// TwinCAT 3 PLC project Untitled1
// ProgramVersion: 3.1.4023.0
// libraries:
//   Tc2_Standard, * (Beckhoff Automation GmbH)
//   Tc2_System, * (Beckhoff Automation GmbH)
//   Tc3_Module, * (Beckhoff Automation GmbH)
// project tree:
//   / PlcTask.TcTTO
//   POUs/ MAIN.TcPOU (not stored)
//   TASK1/ G_Task1.TcGVL, P_Task1.TcPOU (not stored), SensorBrand.TcDUT (not stored)
//   TASK2/ F_DegToRad.TcPOU, F_UpdateParameter2.TcPOU, G_Task2.TcGVL, F_UpdateParameter.TcPOU, P_Task2.TcPOU, ST_MotorParameters.TcDUT, ST_Timer.TcDUT

CONFIGURATION Untitled1
    RESOURCE PLC ON TwinCAT3
        TASK PlcTask(INTERVAL := T#10ms, PRIORITY := 20);
        PROGRAM MAIN WITH PlcTask : MAIN;
    END_RESOURCE
END_CONFIGURATION

// ---- TASK2/ST_MotorParameters.TcDUT
TYPE ST_MotorParameters :
STRUCT
	fMaxMotorSpeed:REAL;
	fMinMotorSpeed:REAL;
END_STRUCT
END_TYPE

// ---- TASK2/ST_Timer.TcDUT
TYPE ST_Timer :
STRUCT
bTimerStart:BOOL;
tTimer:TIME;
bTimerOn:BOOL;
tEllapsedTime:TIME;
END_STRUCT
END_TYPE

// ---- TASK1/G_Task1.TcGVL
{attribute 'qualified_only'}
VAR_GLOBAL
dtvariable:DATE_AND_TIME:=DT#2023-02-07-14:01:20;

tTid:TIME:=T#5S;
aDatoArray:ARRAY[1..4]OF DATE:=[D#2023-02-07, D#2023-02-08,D#2023-02-09,D#2023-02-10];
eSensor1:SensorBrand;
bTimerStart:BOOL;
tTimer:TIME:=T#10S;
bTimerOn:BOOL;
tEllapsedTime:TIME;
END_VAR

// ---- TASK2/G_Task2.TcGVL
{attribute 'qualified_only'}
VAR_GLOBAL
	stTimer2 : ST_Timer:=(tTimer:=T#5S);
	fMotorPosDeg:REAL;
	fMototPosRad:REAL;
	stMotorParametrs:ST_MotorParameters;
	stMotorParameters2:ST_MotorParameters;
	
END_VAR

// ---- TASK2/F_DegToRad.TcPOU
FUNCTION F_DegToRad : REAL
VAR_INPUT
	fDegree:LREAL;
END_VAR
VAR
END_VAR

F_DegToRad:=fDegree*(3.14/180);

END_FUNCTION

// ---- TASK2/F_UpdateParameter2.TcPOU
FUNCTION F_UpdateParameter2 
VAR_INPUT
	bUpdateValue:BOOL;
	fNewValue:REAL;
	stMotorParameter:REFERENCE TO ST_MotorParameters;
END_VAR
VAR
END_VAR

IF bUpdateValue THEN
	stMotorParameter.fMaxMotorSpeed:=fNewValue;
ELSE
	stMotorParameter.fMaxMotorSpeed:=stMotorParameter.fMaxMotorSpeed;
END_IF

END_FUNCTION

// ---- TASK2/F_UpdateParameter.TcPOU
FUNCTION F_UpdateParameter 
VAR_INPUT
	bUpdateValue:BOOL;
	fNewValue:REAL;
	stMotorParameter:ST_MotorParameters;
END_VAR
VAR
END_VAR

IF bUpdateValue THEN
	stMotorParameter.fMaxMotorSpeed:=fNewValue;
ELSE
	stMotorParameter.fMaxMotorSpeed:=stMotorParameter.fMaxMotorSpeed;
END_IF

END_FUNCTION

// ---- TASK2/P_Task2.TcPOU
PROGRAM P_Task2
VAR
	fbTof:TOF;
	fbRTrig:R_TRIG;
	bUpdateMotorSpeed:BOOL;
	fNewValue:REAL;
END_VAR

fbTof (IN:=G_Task2.stTimer2.bTimerStart,
	  PT:=G_Task2.stTimer2.tTimer,
	  ET =>G_Task2.stTimer2.tEllapsedTime,
	  Q =>G_Task2.stTimer2.bTimerOn
	  
	);

G_Task2.fMototPosRad:=F_DegToRad(G_Task2.fMotorPosDeg);
fbRTrig(CLK:=bUpdateMotorSpeed);
F_UpdateParameter(bUpdateValue:=fbRTrig.Q, fNewValue:=fNewValue,stMotorParameter:=G_Task2.stMotorParametrs);
F_UpdateParameter2(bUpdateValue:=fbRTrig.Q, fNewValue:=fNewValue,stMotorParameter:=G_Task2.stMotorParameters2);

END_PROGRAM
